# B&R Automation Studio project NS0453Palletizer
Automation Studio 4.12.2.93; technology packages: mapp 5.22.1, mappCockpit 5.22.0, mappMotion 5.22.2, mappView 5.22.1

## Configuration X20CP1586

CPU X20CP1586, AutomationRuntime G4.93, Build 4.1.2, Safety 0.0, Vc 

### Task classes (Cpu.sw)
```
DataObjects: McAcpSys
NcDataObjects: McDriveLog
Binaries: McAcpDrv, udbdef, McAcpSim, mvLoader, arflatprv, TCData, mCoWebSc, McMechSys, FWRules, arcoal, arsvcreg, Settings, iomap, Config_3, Config_4, Role, ashwac, Hierarchy, asfw, Config_5, sysconf, Config_2, arconfig, Config_1, ashwd, User
Libraries: McBase, MpRobotics, McAxGroup, MpBase, McPathGen, McAxis, McProgInt, McAcpAx, CoTrace, AsZip, FileIO, runtime, MpAxis, MpAlarmX, astime, MpServer, MpFile, asarprof, asieccon, asarlog, asio, asmem, asepl, brsystem, dataobj, arssl, sys_lib, powerlnk
```

### Hardware
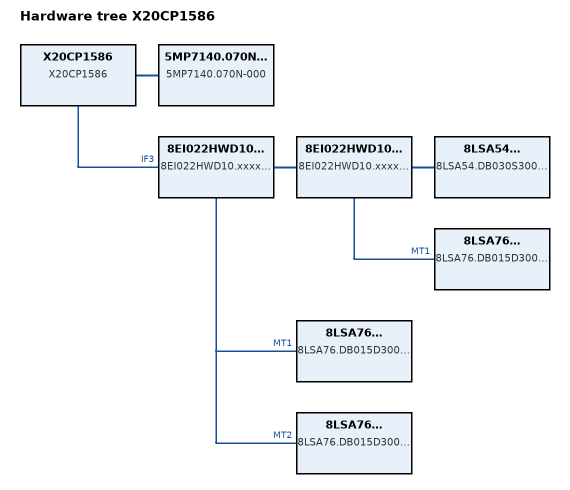
```
5MP7140.070N-000 : 5MP7140.070N-000 v1.1.1.0  [ETH1 -> X20CP1586.IF2 [Cable Type=PowerlinkCable, Length=10, Version=1.0.0.3]]
  Terminal = true
  Startmode = 2
  Mode = Manual
  InternetAddress = 192.168.1.12
  DefaultGateway = 192.168.1.10
  Subnetmask = 255.255.255.0
  PasswordVNCEncrypted = 
  SelectedFavoriteWeb = 192.168.1.10
  PasswordCIFSEncrypted = 
  PasswordServiceEncrypted = 
  VncKeyMappingFile = 
  VncPortNumber = 5901
8EI022HWD10.xxxx-1 : 8EI022HWD10.xxxx-1 v2.3.1.1  [PLK1 -> X20CP1586.IF3 (NodeNumber=1) [Cable Type=PowerlinkCable, Length=10, Version=1.0.0.3]; PLK2 -> 8EI022HWD10.xxxx-1a.PLK1 (NodeNumber=1) [Cable Type=PowerlinkCable, Length=10, Version=1.0.0.3]; MT2 -> 8LSA76.DB015D300-3a.MT]
  EnableDNA = on
  DriveConfiguration/Module:
    McAcoposTypeID = AcoposP3DConfig
    ActivateACOPOSSimulationOnPLC = 0
  DriveConfiguration/Encoder/EncoderX41:
    InterfaceType = EnDat
  DriveConfiguration/Encoder/EncoderX42:
    InterfaceType = EnDat
  DriveConfiguration/Channel[1]/RealAxis:
    AxisReference = gAxisQ1
    MechanicalElementsIsInvisible = 0
  DriveConfiguration/Channel[1]/RealAxis/MechanicalElements/Gearbox:
    InputIsReadOnly = 0
    Input = 1
    OutputIsReadOnly = 0
    Output = 1
  DriveConfiguration/Channel[1]/RealAxis/MechanicalElements/RotaryToLinearTransformation:
    ReferenceDistanceIsReadOnly = 0
    ReferenceDistance = 1
  DriveConfiguration/Channel[1]/RealAxis/Controller:
    ModeIsReadOnly = 0
    Mode = PositionController
  DriveConfiguration/Channel[1]/RealAxis/Controller/Mode/Position:
    ProportionalGain = 50.0
    IntegrationTime = 0.0
    PredictionTime = 0.0004
    TotalDelayTime = 0.0004
  DriveConfiguration/Channel[1]/RealAxis/Controller/Mode/Speed:
    ProportionalGainIsReadOnly = 0
    ProportionalGain = 2.0
    IntegrationTimeIsReadOnly = 0
    IntegrationTime = 0.0
    FilterTimeIsReadOnly = 0
    FilterTime = 0.0
  DriveConfiguration/Channel[1]/RealAxis/Controller/Mode/LoopFilters:
    LoopFilterXIsReadOnly = 0
    LoopFilter1 = NotUsed
    LoopFilter2 = NotUsed
    LoopFilter3 = NotUsed
  DriveConfiguration/Channel[1]/RealAxis/Homing:
    ModeIsReadOnly = 0
    Mode = Direct
  DriveConfiguration/Channel[1]/RealAxis/Homing/Mode:
    Position = 0.0
    ReferencePulse = NotUsed
  DriveConfiguration/Channel[1]/RealAxis/Homing:
    RestorePositionVariable = 
  DriveConfiguration/Channel[1]/RealAxis/StopReaction:
    QuickstopIsReadOnly = 0
    Quickstop = DecelerationLimit
    DriveErrorIsReadOnly = 0
    DriveError = DecelerationLimit
  DriveConfiguration/Channel[1]/RealAxis/MovementErrorLimits:
    PositionError = 100
    VelocityErrorMonitoring = Automatic1
  DriveConfiguration/Channel[1]/RealAxis:
    JerkFilterIsReadOnly = 0
    JerkFilter = NotUsed
  DriveConfiguration/Channel[1]/RealAxis/DigitalInputs/HomingSwitch:
    SourceIsReadOnly = 0
    Source = NotUsed
    Level = High
  DriveConfiguration/Channel[1]/RealAxis/DigitalInputs/PositiveLimitSwitch:
    SourceIsReadOnly = 0
    Source = NotUsed
    Level = High
  DriveConfiguration/Channel[1]/RealAxis/DigitalInputs/NegativeLimitSwitch:
    SourceIsReadOnly = 0
    Source = NotUsed
    Level = High
  DriveConfiguration/Channel[1]/RealAxis/DigitalInputs/Trigger1:
    Source = X8Trigger1
    Level = High
  DriveConfiguration/Channel[1]/RealAxis/DigitalInputs/Trigger2:
    Source = X8Trigger2
    Level = High
  DriveConfiguration/Channel[1]/RealAxis/DigitalInputs/Quickstop:
    Input = Trigger2
  DriveConfiguration/Channel[1]/RealAxis/Simulation:
    SimulationModeOnPLC = SetValueGeneration
    SimulationModeOnACOPOS = NotUsed
  DriveConfiguration/Channel[1]:
    ExternalEncoderAxis = NotUsed
  DriveConfiguration/Channel[2]/RealAxis:
    AxisReference = gAxisQ2
    MechanicalElementsIsInvisible = 0
  DriveConfiguration/Channel[2]/RealAxis/MechanicalElements/Gearbox:
    InputIsReadOnly = 0
    Input = 1
    OutputIsReadOnly = 0
    Output = 1
  DriveConfiguration/Channel[2]/RealAxis/MechanicalElements/RotaryToLinearTransformation:
    ReferenceDistanceIsReadOnly = 0
    ReferenceDistance = 1
  DriveConfiguration/Channel[2]/RealAxis/Controller:
    ModeIsReadOnly = 0
    Mode = PositionController
  DriveConfiguration/Channel[2]/RealAxis/Controller/Mode/Position:
    ProportionalGain = 50.0
    IntegrationTime = 0.0
    PredictionTime = 0.0004
    TotalDelayTime = 0.0004
  DriveConfiguration/Channel[2]/RealAxis/Controller/Mode/Speed:
    ProportionalGainIsReadOnly = 0
    ProportionalGain = 2.0
    IntegrationTimeIsReadOnly = 0
    IntegrationTime = 0.0
    FilterTimeIsReadOnly = 0
    FilterTime = 0.0
  DriveConfiguration/Channel[2]/RealAxis/Controller/Mode/LoopFilters:
    LoopFilterXIsReadOnly = 0
    LoopFilter1 = NotUsed
    LoopFilter2 = NotUsed
    LoopFilter3 = NotUsed
  DriveConfiguration/Channel[2]/RealAxis/Homing:
    ModeIsReadOnly = 0
    Mode = Direct
  DriveConfiguration/Channel[2]/RealAxis/Homing/Mode:
    Position = 0.0
    ReferencePulse = NotUsed
  DriveConfiguration/Channel[2]/RealAxis/Homing:
    RestorePositionVariable = 
  DriveConfiguration/Channel[2]/RealAxis/StopReaction:
    QuickstopIsReadOnly = 0
    Quickstop = DecelerationLimit
    DriveErrorIsReadOnly = 0
    DriveError = DecelerationLimit
  DriveConfiguration/Channel[2]/RealAxis/MovementErrorLimits:
    PositionError = 100
    VelocityErrorMonitoring = Automatic1
  DriveConfiguration/Channel[2]/RealAxis:
    JerkFilterIsReadOnly = 0
    JerkFilter = NotUsed
  DriveConfiguration/Channel[2]/RealAxis/DigitalInputs/HomingSwitch:
    SourceIsReadOnly = 0
    Source = NotUsed
    Level = High
  DriveConfiguration/Channel[2]/RealAxis/DigitalInputs/PositiveLimitSwitch:
    SourceIsReadOnly = 0
    Source = NotUsed
    Level = High
  DriveConfiguration/Channel[2]/RealAxis/DigitalInputs/NegativeLimitSwitch:
    SourceIsReadOnly = 0
    Source = NotUsed
    Level = High
  DriveConfiguration/Channel[2]/RealAxis/DigitalInputs/Trigger1:
    Source = X8Trigger1
    Level = High
  DriveConfiguration/Channel[2]/RealAxis/DigitalInputs/Trigger2:
    Source = X8Trigger2
    Level = High
  DriveConfiguration/Channel[2]/RealAxis/DigitalInputs/Quickstop:
    Input = Trigger2
  DriveConfiguration/Channel[2]/RealAxis/Simulation:
    SimulationModeOnPLC = SetValueGeneration
    SimulationModeOnACOPOS = NotUsed
  DriveConfiguration/Channel[2]:
    ExternalEncoderAxis = NotUsed
8EI022HWD10.xxxx-1a : 8EI022HWD10.xxxx-1 v2.3.1.1  [PLK1 -> 8EI022HWD10.xxxx-1.PLK2 (NodeNumber=2) [Cable Type=PowerlinkCable, Length=10, Version=1.0.0.3]; MT2 -> 8LSA54.DB030S300-3.MT]
  EnableDNA = on
  DriveConfiguration/Module:
    McAcoposTypeID = AcoposP3DConfig
    ActivateACOPOSSimulationOnPLC = 0
  DriveConfiguration/Encoder/EncoderX41:
    InterfaceType = EnDat
  DriveConfiguration/Encoder/EncoderX42:
    InterfaceType = EnDat
  DriveConfiguration/Channel[1]/RealAxis:
    AxisReference = gAxisQ3
    MechanicalElementsIsInvisible = 0
  DriveConfiguration/Channel[1]/RealAxis/MechanicalElements/Gearbox:
    InputIsReadOnly = 0
    Input = 1
    OutputIsReadOnly = 0
    Output = 1
  DriveConfiguration/Channel[1]/RealAxis/MechanicalElements/RotaryToLinearTransformation:
    ReferenceDistanceIsReadOnly = 0
    ReferenceDistance = 1
  DriveConfiguration/Channel[1]/RealAxis/Controller:
    ModeIsReadOnly = 0
    Mode = PositionController
  DriveConfiguration/Channel[1]/RealAxis/Controller/Mode/Position:
    ProportionalGain = 50.0
    IntegrationTime = 0.0
    PredictionTime = 0.0004
    TotalDelayTime = 0.0004
  DriveConfiguration/Channel[1]/RealAxis/Controller/Mode/Speed:
    ProportionalGainIsReadOnly = 0
    ProportionalGain = 2.0
    IntegrationTimeIsReadOnly = 0
    IntegrationTime = 0.0
    FilterTimeIsReadOnly = 0
    FilterTime = 0.0
  DriveConfiguration/Channel[1]/RealAxis/Controller/Mode/LoopFilters:
    LoopFilterXIsReadOnly = 0
    LoopFilter1 = NotUsed
    LoopFilter2 = NotUsed
    LoopFilter3 = NotUsed
  DriveConfiguration/Channel[1]/RealAxis/Homing:
    ModeIsReadOnly = 0
    Mode = Direct
  DriveConfiguration/Channel[1]/RealAxis/Homing/Mode:
    Position = 0.0
    ReferencePulse = NotUsed
  DriveConfiguration/Channel[1]/RealAxis/Homing:
    RestorePositionVariable = 
  DriveConfiguration/Channel[1]/RealAxis/StopReaction:
    QuickstopIsReadOnly = 0
    Quickstop = DecelerationLimit
    DriveErrorIsReadOnly = 0
    DriveError = DecelerationLimit
  DriveConfiguration/Channel[1]/RealAxis/MovementErrorLimits:
    PositionError = 100
    VelocityErrorMonitoring = Automatic1
  DriveConfiguration/Channel[1]/RealAxis:
    JerkFilterIsReadOnly = 0
    JerkFilter = NotUsed
  DriveConfiguration/Channel[1]/RealAxis/DigitalInputs/HomingSwitch:
    SourceIsReadOnly = 0
    Source = NotUsed
    Level = High
  DriveConfiguration/Channel[1]/RealAxis/DigitalInputs/PositiveLimitSwitch:
    SourceIsReadOnly = 0
    Source = NotUsed
    Level = High
  DriveConfiguration/Channel[1]/RealAxis/DigitalInputs/NegativeLimitSwitch:
    SourceIsReadOnly = 0
    Source = NotUsed
    Level = High
  DriveConfiguration/Channel[1]/RealAxis/DigitalInputs/Trigger1:
    Source = X8Trigger1
    Level = High
  DriveConfiguration/Channel[1]/RealAxis/DigitalInputs/Trigger2:
    Source = X8Trigger2
    Level = High
  DriveConfiguration/Channel[1]/RealAxis/DigitalInputs/Quickstop:
    Input = Trigger2
  DriveConfiguration/Channel[1]/RealAxis/Simulation:
    SimulationModeOnPLC = SetValueGeneration
    SimulationModeOnACOPOS = NotUsed
  DriveConfiguration/Channel[1]:
    ExternalEncoderAxis = NotUsed
  DriveConfiguration/Channel[2]/RealAxis:
    AxisReference = gAxisQ4
    MechanicalElementsIsInvisible = 0
  DriveConfiguration/Channel[2]/RealAxis/MechanicalElements/Gearbox:
    InputIsReadOnly = 0
    Input = 1
    OutputIsReadOnly = 0
    Output = 1
  DriveConfiguration/Channel[2]/RealAxis/MechanicalElements/RotaryToLinearTransformation:
    ReferenceDistanceIsReadOnly = 0
    ReferenceDistance = 1
  DriveConfiguration/Channel[2]/RealAxis/Controller:
    ModeIsReadOnly = 0
    Mode = PositionController
  DriveConfiguration/Channel[2]/RealAxis/Controller/Mode/Position:
    ProportionalGain = 50.0
    IntegrationTime = 0.0
    PredictionTime = 0.0004
    TotalDelayTime = 0.0004
  DriveConfiguration/Channel[2]/RealAxis/Controller/Mode/Speed:
    ProportionalGainIsReadOnly = 0
    ProportionalGain = 2.0
    IntegrationTimeIsReadOnly = 0
    IntegrationTime = 0.0
    FilterTimeIsReadOnly = 0
    FilterTime = 0.0
  DriveConfiguration/Channel[2]/RealAxis/Controller/Mode/LoopFilters:
    LoopFilterXIsReadOnly = 0
    LoopFilter1 = NotUsed
    LoopFilter2 = NotUsed
    LoopFilter3 = NotUsed
  DriveConfiguration/Channel[2]/RealAxis/Homing:
    ModeIsReadOnly = 0
    Mode = Direct
  DriveConfiguration/Channel[2]/RealAxis/Homing/Mode:
    Position = 0.0
    ReferencePulse = NotUsed
  DriveConfiguration/Channel[2]/RealAxis/Homing:
    RestorePositionVariable = 
  DriveConfiguration/Channel[2]/RealAxis/StopReaction:
    QuickstopIsReadOnly = 0
    Quickstop = DecelerationLimit
    DriveErrorIsReadOnly = 0
    DriveError = DecelerationLimit
  DriveConfiguration/Channel[2]/RealAxis/MovementErrorLimits:
    PositionError = 100
    VelocityErrorMonitoring = Automatic1
  DriveConfiguration/Channel[2]/RealAxis:
    JerkFilterIsReadOnly = 0
    JerkFilter = NotUsed
  DriveConfiguration/Channel[2]/RealAxis/DigitalInputs/HomingSwitch:
    SourceIsReadOnly = 0
    Source = NotUsed
    Level = High
  DriveConfiguration/Channel[2]/RealAxis/DigitalInputs/PositiveLimitSwitch:
    SourceIsReadOnly = 0
    Source = NotUsed
    Level = High
  DriveConfiguration/Channel[2]/RealAxis/DigitalInputs/NegativeLimitSwitch:
    SourceIsReadOnly = 0
    Source = NotUsed
    Level = High
  DriveConfiguration/Channel[2]/RealAxis/DigitalInputs/Trigger1:
    Source = X8Trigger1
    Level = High
  DriveConfiguration/Channel[2]/RealAxis/DigitalInputs/Trigger2:
    Source = X8Trigger2
    Level = High
  DriveConfiguration/Channel[2]/RealAxis/DigitalInputs/Quickstop:
    Input = Trigger2
  DriveConfiguration/Channel[2]/RealAxis/Simulation:
    SimulationModeOnPLC = SetValueGeneration
    SimulationModeOnACOPOS = NotUsed
  DriveConfiguration/Channel[2]:
    ExternalEncoderAxis = NotUsed
8LSA54.DB030S300-3 : 8LSA54.DB030S300-3 v2.2.1.0  [MT -> 8EI022HWD10.xxxx-1a.MT2]
  M1/MotorParameters:
    MOTOR_AMB_TEMP_RATED = 40
8LSA76.DB015D300-3 : 8LSA76.DB015D300-3 v2.2.0.0  [MT -> 8EI022HWD10.xxxx-1.MT1]
  M1/MotorParameters:
    MOTOR_AMB_TEMP_RATED = 40
8LSA76.DB015D300-3a : 8LSA76.DB015D300-3 v2.2.0.0  [MT -> 8EI022HWD10.xxxx-1.MT2]
  M1/MotorParameters:
    MOTOR_AMB_TEMP_RATED = 40
8LSA76.DB015D300-3b : 8LSA76.DB015D300-3 v2.2.0.0  [MT -> 8EI022HWD10.xxxx-1a.MT1]
  M1/MotorParameters:
    MOTOR_AMB_TEMP_RATED = 40
X20CP1586 : X20CP1586 v1.10.0.0
  Connector IF2:
    ActivateDevice = 1
    Mode = Manual
    InternetAddress = 192.168.1.10
    SubnetMask = 255.255.255.0
    ActivateSnmp = 2
  Connector IF3:
    CycleTime = 400
    Channel1
    ChannelID1 = McAcpBroadcast
    ChannelType1 = OCTET[96]
  ConfigurationID = NS0453RobotPack_Config1
  UserPartitionSize = 200
  Simulation = 1
  TimerDeviceType = EPLX2X
  TimerDevice = X20CP1586.IF3
  TaskClassIdleTime = 2000
  Cyclic1Duration = 800
  Cyclic1Tolerance = 0
  Cyclic1Output = 1
  FileDevice1
  FileDeviceName1 = USER
  FileDevicePath1 = USER_PATH
  FileDevice2
  FileDeviceName2 = Robot_FTP
  FileDevicePath2 = F:\RobotPrg\
  FtpUser1
  FtpUsername1 = Robot
  FtpUserPassword1 = ZoXDR9dI9SfvDHy33U2CpOF+f1SFYYRLOF1GTOMGY30=
  FtpUserSalt1 = nNkeD+gM
  FTPAccessRight1 = 0
  FTPdevice1 = ALL
  ActivateOpcUa = 1
  OpcUaInformationModels_PV_Version = 1
```

### IoMap.iom - X20CP1586/IoMap.iom
```iecst
VAR_CONFIG
	::gRobotControl.IHMCmd.Input.SpeedUp AT %ID."5MP7140.070N-000".Key1;
	::gRobotControl.IHMCmd.Input.SpeedDown AT %ID."5MP7140.070N-000".Key2;
	::gRobotControl.IHMCmd.Input.F1 AT %ID."5MP7140.070N-000".Key3;
	::gRobotControl.IHMCmd.Input.F2 AT %ID."5MP7140.070N-000".Key4;
	::gRobotControl.IHMCmd.Input.F3 AT %ID."5MP7140.070N-000".Key5;
	::gRobotControl.IHMCmd.Input.F4 AT %ID."5MP7140.070N-000".Key6;
	::gRobotControl.IHMCmd.Input.F5 AT %ID."5MP7140.070N-000".Key7;
	::gRobotControl.IHMCmd.Input.F6 AT %ID."5MP7140.070N-000".Key8;
	::gRobotControl.IHMCmd.Input.ApplicationScreen AT %ID."5MP7140.070N-000".Key9;
	::gRobotControl.IHMCmd.Input.ProjectScreen AT %ID."5MP7140.070N-000".Key10;
	::gRobotControl.IHMCmd.Input.PositionScreen AT %ID."5MP7140.070N-000".Key11;
	::gRobotControl.IHMCmd.Input.VariableMonitor AT %ID."5MP7140.070N-000".Key12;
	::gRobotControl.IHMCmd.Input.Start AT %ID."5MP7140.070N-000".Key13;
	::gRobotControl.IHMCmd.Input.Stop AT %ID."5MP7140.070N-000".Key14;
	::gRobotControl.IHMCmd.Input.CustomerSetting AT %ID."5MP7140.070N-000".Key15;
	::gRobotControl.IHMCmd.Input.Cancel AT %ID."5MP7140.070N-000".Key16;
	::gRobotControl.IHMCmd.Input.Plane2 AT %ID."5MP7140.070N-000".Key17;
	::gRobotControl.IHMCmd.Input.AlarmScreen AT %ID."5MP7140.070N-000".Key18;
	::gRobotControl.IHMCmd.Output.Run AT %QD."5MP7140.070N-000".Led0;
	::gRobotControl.IHMCmd.Output.Error AT %QD."5MP7140.070N-000".Led1;
	::gRobotControl.IHMCmd.Output.Motion AT %QD."5MP7140.070N-000".Led2;
	::gRobotControl.IHMCmd.Output.Process AT %QD."5MP7140.070N-000".Led3;
	::gRobotControl.IHMCmd.Output.Plane2 AT %QD."5MP7140.070N-000".Led4;
	::gRobotControl.IHMCmd.Input.Manual AT %ID."5MP7140.070N-000".Keyswitch0;
	::gRobotControl.IHMCmd.Input.Automatic AT %ID."5MP7140.070N-000".Keyswitch1;
	::gRobotControl.IHMCmd.Input.Ctrl  AT %ID."5MP7140.070N-000".Key19;
END_VAR
```

### Config_1.axesgroup - X20CP1586/mappMotion/4AxesRoboarmA/Config_1.axesgroup
```
Element g4AxRobA (Type=axesgroup)
  Type = PathGenAxesGroup
    ProcessingTaskClass = 255
    License = 1
    PhysicalAxes:
      JointAxes:
        JointAxisAxisRefIsReadOnly = 0
        JointAxis[1]:
          Name = Q1
          AxisRef = gAxisQ1
        JointAxis[2]:
          Name = Q2
          AxisRef = gAxisQ2
        JointAxis[3]:
          Name = Q3
          AxisRef = gAxisQ3
        JointAxis[4]:
          Name = Q4
          AxisRef = gAxisQ4
    MechanicalSystem:
      MechSysRefIsReadOnly = 0
      MechSysRef = MechSys_4AxRobA
    BasicSettings:
      ModalDataBehaviour = ResetToDefault
      GeometryPlanning:
        TCPResolutionIsReadOnly = 0
        TCPResolution:
          LengthResolution = 0.001
          AngleResolution = 0.001
        Rounding:
          PathDistance = 0.0
          SymmetricRounding = Yes
          LastSegment = Half
        RoundingMode = Standard
        MaxCornerDeviation = 0.0
        MaxTangentialTransitionDeviation = 0.0
        MaxRadiusDeviation = 0.001
        WorkingPlane = XY
      TrajectoryPlanningIsReadOnly = 0
      TrajectoryPlanning = Basic
        LimitCheckResolutionIsReadOnly = 0
        LimitCheckResolution = UserDefinedTime
          TimeIsReadOnly = 0
          Time = 0.01
        BufferTime = UserDefinedTime
          Time = 0.1
        BarrierParametrization = JointCoordinates
      Miscellaneous:
        NonMovementsLimit = NotUsed
        TimeStretchOverride:
          JerkSuppression = NotUsed
    AxesGroupFeatures:
      FeatureRef[1] = Feature_Programs
      FeatureRef[2] = Feature_Jogging
  Alarms = MpAlarmX
```

### Config_2.axis - X20CP1586/mappMotion/4AxesRoboarmA/Config_2.axis
```
Element gAxisQ1 (Type=axis)
  BaseTypeIsReadOnly = 0
  BaseType = RotaryBounded
    MeasurementUnitIsReadOnly = 0
    MeasurementUnit = 17476
    MeasurementResolutionIsReadOnly = 0
    MeasurementResolution = 0.01
    CountDirectionIsReadOnly = 0
    CountDirection = Standard
  MovementLimitsIsReadOnly = 0
  MovementLimits = Internal
    Position:
      LowerLimitMin = -1.79769313486231E308
      UpperLimitMax = 1.79769313486231E308
      LowerLimit = -1000.0
      UpperLimit = 1000.0
    VelocityIsReadOnly = 0
    Velocity:
      VelocityMax = 3.4E38
      Velocity = 10000
    AccelerationIsReadOnly = 0
    Acceleration:
      AccelerationMax = 3.4E38
      Acceleration = 5000
    DecelerationIsReadOnly = 0
    Deceleration:
      DecelerationMax = 3.4E38
      Deceleration = 5000
  Alarms = MpAlarmX
Element gAxisQ2 (Type=axis)
  BaseTypeIsReadOnly = 0
  BaseType = RotaryBounded
    MeasurementUnitIsReadOnly = 0
    MeasurementUnit = 17476
    MeasurementResolutionIsReadOnly = 0
    MeasurementResolution = 0.01
    CountDirectionIsReadOnly = 0
    CountDirection = Standard
  MovementLimitsIsReadOnly = 0
  MovementLimits = Internal
    Position:
      LowerLimitMin = -1.79769313486231E308
      UpperLimitMax = 1.79769313486231E308
      LowerLimit = -1000.0
      UpperLimit = 1000.0
    VelocityIsReadOnly = 0
    Velocity:
      VelocityMax = 3.4E38
      Velocity = 1000
    AccelerationIsReadOnly = 0
    Acceleration:
      AccelerationMax = 3.4E38
      Acceleration = 5000
    DecelerationIsReadOnly = 0
    Deceleration:
      DecelerationMax = 3.4E38
      Deceleration = 5000
  Alarms = MpAlarmX
Element gAxisQ3 (Type=axis)
  BaseTypeIsReadOnly = 0
  BaseType = RotaryBounded
    MeasurementUnitIsReadOnly = 0
    MeasurementUnit = 17476
    MeasurementResolutionIsReadOnly = 0
    MeasurementResolution = 0.01
    CountDirectionIsReadOnly = 0
    CountDirection = Standard
  MovementLimitsIsReadOnly = 0
  MovementLimits = Internal
    Position:
      LowerLimitMin = -1.79769313486231E308
      UpperLimitMax = 1.79769313486231E308
      LowerLimit = -1000.0
      UpperLimit = 1000.0
    VelocityIsReadOnly = 0
    Velocity:
      VelocityMax = 3.4E38
      Velocity = 1000
    AccelerationIsReadOnly = 0
    Acceleration:
      AccelerationMax = 3.4E38
      Acceleration = 5000
    DecelerationIsReadOnly = 0
    Deceleration:
      DecelerationMax = 3.4E38
      Deceleration = 5000
  Alarms = MpAlarmX
Element gAxisQ4 (Type=axis)
  BaseTypeIsReadOnly = 0
  BaseType = RotaryBounded
    MeasurementUnitIsReadOnly = 0
    MeasurementUnit = 17476
    MeasurementResolutionIsReadOnly = 0
    MeasurementResolution = 0.01
    CountDirectionIsReadOnly = 0
    CountDirection = Standard
  MovementLimitsIsReadOnly = 0
  MovementLimits = Internal
    Position:
      LowerLimitMin = -1.79769313486231E308
      UpperLimitMax = 1.79769313486231E308
      LowerLimit = -1000.0
      UpperLimit = 1000.0
    VelocityIsReadOnly = 0
    Velocity:
      VelocityMax = 3.4E38
      Velocity = 1000
    AccelerationIsReadOnly = 0
    Acceleration:
      AccelerationMax = 3.4E38
      Acceleration = 5000
    DecelerationIsReadOnly = 0
    Deceleration:
      DecelerationMax = 3.4E38
      Deceleration = 5000
  Alarms = MpAlarmX
```

### Config_3.mechanicalsystem - X20CP1586/mappMotion/4AxesRoboarmA/Config_3.mechanicalsystem
```
Element MechSys_4AxRobA (Type=mechanicalsystem)
  TypeIsReadOnly = 0
  Type = 4AxesRoboarm
    SubtypeIsReadOnly = 0
    Subtype = 4AxesRoboarmA
      SceneViewerObject = NotUsed
      DescriptionIsReadOnly = 0
      Description = Standard
        Dimensions:
          TranslationFromBaseToQ1IsReadOnly = 0
          TranslationFromBaseToQ1:
            X = 0.0
            Y = 0.0
            Z = 350.0
          TranslationFromQ1ToQ2IsReadOnly = 0
          TranslationFromQ1ToQ2:
            X = 400.0
            Y = 0.0
            Z = 400.0
          TranslationFromQ2ToQ3IsReadOnly = 0
          TranslationFromQ2ToQ3:
            X = 0.0
            Y = 0.0
            Z = 1175.0
          TranslationFromQ3ToPQ1IsReadOnly = 0
          TranslationFromQ3ToPQ1:
            X = 1360.0
            Y = 0.0
            Z = 0.0
          TranslationFromPQ1ToQ4IsReadOnly = 0
          TranslationFromPQ1ToQ4:
            X = 250.0
            Y = 0.0
            Z = -250.0
          TranslationFromQ4ToFlangeIsReadOnly = 0
          TranslationFromQ4ToFlange:
            X = 0.0
            Y = 0.0
            Z = -50.0
        Offsets:
          JointAxisIsReadOnly = 0
          JointAxis[1] = 0.0
          JointAxis[2] = 0.0
          JointAxis[3] = 0.0
          JointAxis[4] = 0.0
        CountDirections:
          JointAxisIsReadOnly = 0
          JointAxis[1] = Standard
          JointAxis[2] = Standard
          JointAxis[3] = Inverse
          JointAxis[4] = Standard
      CoordinatesNames = Default
        XCoordinateName = X
        YCoordinateName = Y
        ZCoordinateName = Z
        CCoordinateName = C
      WireFrameModelIsReadOnly = 0
      WireFrameModel = Standard
        Q1ToQ2IsReadOnly = 0
        Q1ToQ2 = ConnectionLine
          DistanceMin = -1.79769313486231E308
          DistanceMax = 1.79769313486231E308
          Distance = 0.0
        Q2ToQ3IsReadOnly = 0
        Q2ToQ3 = ConnectionLine
          DistanceMin = -1.79769313486231E308
          DistanceMax = 1.79769313486231E308
          Distance = 0.0
        Q3ToPQ1IsReadOnly = 0
        Q3ToPQ1 = ConnectionLine
          DistanceMin = -1.79769313486231E308
          DistanceMax = 1.79769313486231E308
          Distance = 0.0
        PQ1ToQ4IsReadOnly = 0
        PQ1ToQ4 = ConnectionLine
          DistanceMin = -1.79769313486231E308
          DistanceMax = 1.79769313486231E308
          Distance = 0.0
        Q4ToFlangeIsReadOnly = 0
        Q4ToFlange = ConnectionLine
          DistanceMin = -1.79769313486231E308
          DistanceMax = 1.79769313486231E308
          Distance = 0.0
        FlangeToTcp = ConnectionLine
          DistanceMin = -1.79769313486231E308
          DistanceMax = 1.79769313486231E308
          Distance = 0.0
      DynamicModel = DynParTable
        TableRef
      InternalDynamicModelIsReadOnly = 0
      InternalDynamicModel = NotUsed
      CouplingsIsInvisible = 0
      Couplings:
        LinearCoupling[1]:
          SourceAxisIsReadOnly = 0
          SourceAxis = 2
          SourceAxisUnitsIsReadOnly = 0
          SourceAxisUnits = 1.0
          TargetJointAxisIsReadOnly = 0
          TargetJointAxis = 3
          TargetJointAxisUnitsIsReadOnly = 0
          TargetJointAxisUnits = -1.0
      JointAxesPositionLimits:
        JointAxisIsReadOnly = 0
        JointAxis[1] = UseAxisLimits
        JointAxis[2] = UseAxisLimits
        JointAxis[3] = UseAxisLimits
        JointAxis[4] = UseAxisLimits
```

### Config_4.axesgroupfeature - X20CP1586/mappMotion/4AxesRoboarmA/Config_4.axesgroupfeature
```
Element Feature_Programs (Type=axesgroupfeature)
  Type = Program
    ModalDataBehaviour = UseAxesGroupSettings
    InitialSettings:
      InterpolationTypes = LinearRapid
      PositionCoordinates = Absolute
      CircleCoordinates = Relative
      JACS_ACSProgramming = JACS
      ContourConnection = Inactive
      ProgrammingUnits = UseAxesGroupSettings
      Feedrates:
        FeedPath = Standard
        FeedCharacteristic = StandardCharacteristic
        FeedType = Feedrate
        FeedReduction = Inactive
        FeedrateValue = 0.0
        InverseFeedrateValue = 0.0
        FeedratePerRevValue = 0.0
    DefaultLanguage = BRGCode
    Location = User
      UserLocation[1]:
        FileDevice = Robot_FTP
Element Feature_Jogging (Type=axesgroupfeature)
  Type = Jogging
```

### Config.mpfilemanager - X20CP1586/mappServices/Config.mpfilemanager
```
Element FileManagement (Type=mpfilemanager)
  FileManager:
    Devices:
      0:
        DeviceName = Robot_FTP
        Text = Robot_FTP
    Access:
      0:
        Folder = *
        Roles:
          0:
            Role = Everyone
            Rights:
              Visible = TRUE
              FolderRead = TRUE
              FileRead = TRUE
              FileEdit = TRUE
              FolderEdit = TRUE
  FileManagerRestrict:
    0:
      Functionality = TextEditor
```

## Logical view

Binary libraries used (declarations not repeated): operator, runtime, astime, AsIecCon, AsZip, FileIO, McBase, MpAxis, McAcpAx, McPathGen 5.22.2, McAxGroup, McAxis, McProgInt 5.22.2, MpBase, MpRobotics 5.22.2, MpFile, MpAlarmX, CoTrace, MpServer 5.22.0

### Global.typ
```iecst
TYPE
	IHMCmdInType : 	STRUCT
		SpeedUp : DINT;
		SpeedDown : DINT;
		Start : DINT;
		Stop : DINT;
		F1 : DINT;
		F2 : DINT;
		F3 : DINT;
		F4 : DINT;
		F5 : DINT;
		F6 : DINT;
		Plane2 : DINT;
		Ctrl : DINT;
		PositionScreen : DINT;
		ProjectScreen : DINT;
		VariableMonitor : DINT;
		CustomerSetting : DINT;
		ApplicationScreen : DINT;
		AlarmScreen : DINT;
		Cancel : DINT;
		Manual : DINT;
		Automatic : DINT;
	END_STRUCT;
	IHMCmdOutType : 	STRUCT
		Run : DINT;
		Error : DINT;
		Motion : DINT;
		Process : DINT;
		Plane2 : DINT;
	END_STRUCT;
	IHMCmdTyoe : 	STRUCT
		Input : IHMCmdInType;
		Output : IHMCmdOutType;
	END_STRUCT;
	RobotControlType : 	STRUCT
		IHMCmd : IHMCmdTyoe;
	END_STRUCT;
	IHMInOutRobotType : 	STRUCT
		Input : IHMInputRobotType;
		Output : IHMOutputRobotType;
	END_STRUCT;
	IHMInputRobotType : 	STRUCT
		ServoOn : DINT; (*Servo Off -> 0 / Servo On -> 1 / Servo fault ->2 *)
		ProgramActive : DINT; (*Program Off -> 0 / Program Active ->1 / Program Fault -> 2*)
		ManualAutomatic : DINT; (*Stop -> 0 / Manual Off -> 1 / Manual Active -> 2 / Manual Fault -> 3 / Automatic Off -> 4 / Automatic Active -> 5 / Automatic Fault -> 6*)
		PorcentVelocity : DINT; (*Velocity in Automatic or Manual *)
		F1F2 : DINT; (*Jog Q1 Inactive-> 0 / Jog Q1 Active-> 1 / Jog Q4 Inactive -> 2 / Jog Q4 Active -> 3 / Jog X Inactive -> 4 / Jog X Active -> 5 / Jog C Inactive -> 6  / Jog C Active -> 6 *)
		F3F4 : DINT; (*Jog Q2 Inactive -> 0 / Jog Q2 Active -> 1 / Jog Y Inactive -> 2 / Jog Y Active -> 3*)
		F5F6 : DINT; (*Jog Q3 Inactive -> 0 / Jog Q3 Active -> 1 / Jog Z Inactive -> 2 / Jog Z Active -> 3*)
		VariableMonitor : DINT; (*Inactive*)
		PositioningScreen : DINT; (*Jog -> 0 / World -> 1 / Tools -> 2*)
		StartStop : DINT; (*Stop -> 0 / Start -> 1*)
		CustomerSettingsServicePage : DINT; (*Inactive*)
		Cancel2Plane : DINT; (*Inactive*)
		Error : DINT; (*Inactive*)
		SecondFunction : BOOL;
		EnableQ4 : BOOL;
		EnableC : BOOL;
	END_STRUCT;
	IHMOutputRobotType : 	STRUCT
		VelocityPercent : DINT;
	END_STRUCT;
END_TYPE
```

### Global.var
```iecst
VAR
	gRobotControl : RobotControlType;
	IHMInOutRobot : IHMInOutRobotType;
	gRoboParametros : MpRoboArm4AxisParType;
END_VAR
```
